// TIA Portal project "conveyer belt system V6.4" (V19)

(* hardware
DEVICE "S71500/ET200MP-Station_1"  S7-1500 station
   slot 0: "Profilschiene_0"  6ES7 590-1***0-0AA0
   slot 1: "PLC_1"  CPU 1511-1 PN  6ES7 511-1AK00-0AB0  V1.8
   slot 2: "AI 8xU/I/RTD/TC ST_1"  AI 8xU/I/RTD/TC ST  6ES7 531-7KF00-0AB0  V2.0
   slot 3: "AI 8xU/I/RTD/TC ST_2"  AI 8xU/I/RTD/TC ST  6ES7 531-7KF00-0AB0  V2.0
   slot 4: "AI 8xU/I/RTD/TC ST_3"  AI 8xU/I/RTD/TC ST  6ES7 531-7KF00-0AB0  V2.0
   slot 5: "AI 8xU/I/RTD/TC ST_4"  AI 8xU/I/RTD/TC ST  6ES7 531-7KF00-0AB0  V2.0
   slot 6: "DI 16x24VDC BA_1"  DI 16x24VDC BA  6ES7 521-1BH10-0AA0  V1.0
DEVICE "HMI_1"  KTP1200 Basic PN
   slot 0: "HMI_1"  KTP1200 Basic PN  6AV2 123-2MB03-0AX0  17.0.0.0
   slot 1: "HMI_RT_2"  KTP1200 Basic PN  6AV2 123-2MB03-0AX0  17.0.0.0
   slot 5: "HMI_1.IE_CP_1"  PROFINET Interface  17.0.0.0
      slot 1: "PROFINET Interface_1"  PROFINET Interface
         slot 1: "Port_1"  Port
*)

// ===== PLC "PLC_1"  CPU 1511-1 PN =====

VAR_GLOBAL   // PLC tag table "Standard-Variablentabelle"
   "Tag_1" AT %I1000.0 : Bool;
   "Tag_2" AT %Q1000.0 : Bool;
   "Tag_3" AT %I1000.1 : Bool;
END_VAR

VAR_GLOBAL   // PLC tag table "control panel"
   "start_button" AT %I0.0 : Bool;
   "reset_button" AT %I0.1 : Bool;
   "stop_button" AT %I0.2 : Bool;
   "emergency_stop" AT %I0.3 : Bool;
   "start_button_light" AT %Q0.0 : Bool;
   "reset_button_light" AT %Q0.1 : Bool;
   "stop_button_light" AT %Q0.2 : Bool;
   "system_start" AT %Q0.3 : Bool;
   "system_fault" AT %Q0.4 : Bool;
   "system_stop" AT %Q0.5 : Bool;
   "sensor_start" AT %I0.7 : Bool;
   "low_power_mode" AT %I0.4 : Bool;
   "sensor_carousel" AT %I1.0 : Bool;
   "carousel_on" AT %I0.5 : Bool;
END_VAR

VAR_GLOBAL   // PLC tag table "conveyor 0"
   "motor+(0)" AT %Q3.7 : Bool;
   "motor-(0)" AT %Q3.6 : Bool;
   "encoder_A(0)" AT %I3.7 : Bool;
   "encoder_B(0)" AT %I3.6 : Bool;
   "sensor(0)" AT %I5.7 : Bool;
END_VAR

VAR_GLOBAL   // PLC tag table "conveyor 1"
   "motor+(1)" AT %Q3.5 : Bool;
   "motor-(1)" AT %Q3.4 : Bool;
   "encoder_A(1)" AT %I3.5 : Bool;
   "encoder_B(1)" AT %I3.4 : Bool;
   "sensor(1)" AT %I5.6 : Bool;
END_VAR

VAR_GLOBAL   // PLC tag table "conveyor 2"
   "motor+(2)" AT %Q3.3 : Bool;
   "motor-(2)" AT %Q3.2 : Bool;
   "encoder_A(2)" AT %I3.3 : Bool;
   "encoder_B(2)" AT %I3.2 : Bool;
   "sensor(2)" AT %I5.5 : Bool;
END_VAR

VAR_GLOBAL   // PLC tag table "conveyor 3"
   "motor+(3)" AT %Q3.1 : Bool;
   "motor-(3)" AT %Q3.0 : Bool;
   "encoder_A(3)" AT %I3.1 : Bool;
   "encoder_B(3)" AT %I3.0 : Bool;
   "sensor(3)" AT %I5.4 : Bool;
END_VAR

VAR_GLOBAL   // PLC tag table "conveyor 4"
   "motor+(4)" AT %Q2.7 : Bool;
   "motor-(4)" AT %Q2.6 : Bool;
   "encoder_A(4)" AT %I2.7 : Bool;
   "encoder_B(4)" AT %I2.6 : Bool;
   "sensor(4)" AT %I5.3 : Bool;
END_VAR

VAR_GLOBAL   // PLC tag table "conveyor 5"
   "motor+(5)" AT %Q2.5 : Bool;
   "motor-(5)" AT %Q2.4 : Bool;
   "encoder_A(5)" AT %I2.5 : Bool;
   "encoder_B(5)" AT %I2.4 : Bool;
   "sensor(5)" AT %I5.2 : Bool;
END_VAR

VAR_GLOBAL   // PLC tag table "conveyor 6"
   "motor+(6)" AT %Q2.3 : Bool;
   "motor-(6)" AT %Q2.2 : Bool;
   "encoder_A(6)" AT %I2.3 : Bool;
   "encoder_B(6)" AT %I2.2 : Bool;
   "sensor(6)" AT %I5.1 : Bool;
END_VAR

DATA_BLOCK "conveyor_0"   // DB1
{ S7_Optimized_Access := 'TRUE' }
VERSION : 0.1
// stored: InstanceOfName conveyor_control
"conveyor_control"
BEGIN
END_DATA_BLOCK

DATA_BLOCK "conveyor_2"   // DB3
{ S7_Optimized_Access := 'TRUE' }
VERSION : 0.1
// stored: InstanceOfName conveyor_control
"conveyor_control"
BEGIN
END_DATA_BLOCK

DATA_BLOCK "conveyor_1"   // DB5
{ S7_Optimized_Access := 'TRUE' }
VERSION : 0.1
// stored: InstanceOfName conveyor_control
"conveyor_control"
BEGIN
END_DATA_BLOCK

DATA_BLOCK "system_control_DB"   // DB6
{ S7_Optimized_Access := 'TRUE' }
VERSION : 0.1
// stored: InstanceOfName system_control
"system_control"
BEGIN
END_DATA_BLOCK

DATA_BLOCK "lamp control_DB"   // DB11
{ S7_Optimized_Access := 'TRUE' }
VERSION : 0.1
// stored: InstanceOfName lamp_control
"lamp_control"
BEGIN
END_DATA_BLOCK

DATA_BLOCK "conveyor_3"   // DB15
{ S7_Optimized_Access := 'TRUE' }
VERSION : 0.1
// stored: InstanceOfName conveyor_control
"conveyor_control"
BEGIN
END_DATA_BLOCK

DATA_BLOCK "conveyor_4"   // DB17
{ S7_Optimized_Access := 'TRUE' }
VERSION : 0.1
// stored: InstanceOfName conveyor_control
"conveyor_control"
BEGIN
END_DATA_BLOCK

DATA_BLOCK "conveyor_5"   // DB19
{ S7_Optimized_Access := 'TRUE' }
VERSION : 0.1
// stored: InstanceOfName conveyor_control
"conveyor_control"
BEGIN
END_DATA_BLOCK

DATA_BLOCK "conveyor_6"   // DB21
{ S7_Optimized_Access := 'TRUE' }
VERSION : 0.1
// stored: InstanceOfName conveyor_control
"conveyor_control"
BEGIN
END_DATA_BLOCK

DATA_BLOCK "standard_parameters"   // DB26
{ S7_Optimized_Access := 'TRUE' }
VERSION : 0.1
   VAR
      "2 meter belt clearance delay" : Time := T#4S;   // need to change to 10s
      "4 meter belt clearance delay" : Time := T#8S;   // need to change to 20s
      "6 meter belt clearance delay" : Time := T#12S;   // need to change to 30s
      "curved belt clearance delay" : Time := T#4S;   // need to change to 10s
   END_VAR
BEGIN
END_DATA_BLOCK

DATA_BLOCK "system_state"   // DB27
{ S7_Optimized_Access := 'TRUE' }
VERSION : 0.1
   VAR
      start_0 : Bool;
      start_1 : Bool;
      all_conveyors_running : Bool;
      some_conveyors_running : Bool;
      "system_start/stop_memory" : Bool;
      fault_flag : Bool;
      low_power_mode : Bool;
      safety_delay : Time;
   END_VAR
BEGIN
END_DATA_BLOCK

FUNCTION_BLOCK "conveyor_control"   // FB1, FBD
{ S7_Optimized_Access := 'TRUE' }
VERSION : 0.1
   VAR_INPUT
      enable_cascade_control : Bool;
      enable_sensor_control : Bool;
      enable_on_delay : Bool;
      enable_off_delay : Bool;
      encoder_A : Bool;
      encoder_B : Bool;
      fault_feedback_in : Bool;
      fault_reset : Bool;
      preceeding_sensor : Bool;
      off_delay : Time;
      on_delay : Time := T#1S;
   END_VAR
   VAR_OUTPUT
      "motor+" : Bool;
      "motor-" : Bool;
      motor_fault : Bool;
      motor_condition : Int;
      fault_feedback_out : Bool;
      remaining_delay : Time;
      running_feedback : Bool;
   END_VAR
   VAR_IN_OUT
      system_fault_flag : Bool;
   END_VAR
   VAR
      encoder_buffer : TOF_TIME;
      encoder_A_edge : R_TRIG;
      encoder_B_edge : R_TRIG;
      fault_buffer : TON_TIME;
      sensor_control_Instance : "sensor_control";
   END_VAR
   VAR RETAIN
      off_delay_instance : TOF_TIME;
      on_delay_instance : TON_TIME;
   END_VAR
BEGIN

REGION Network 1: sensor control
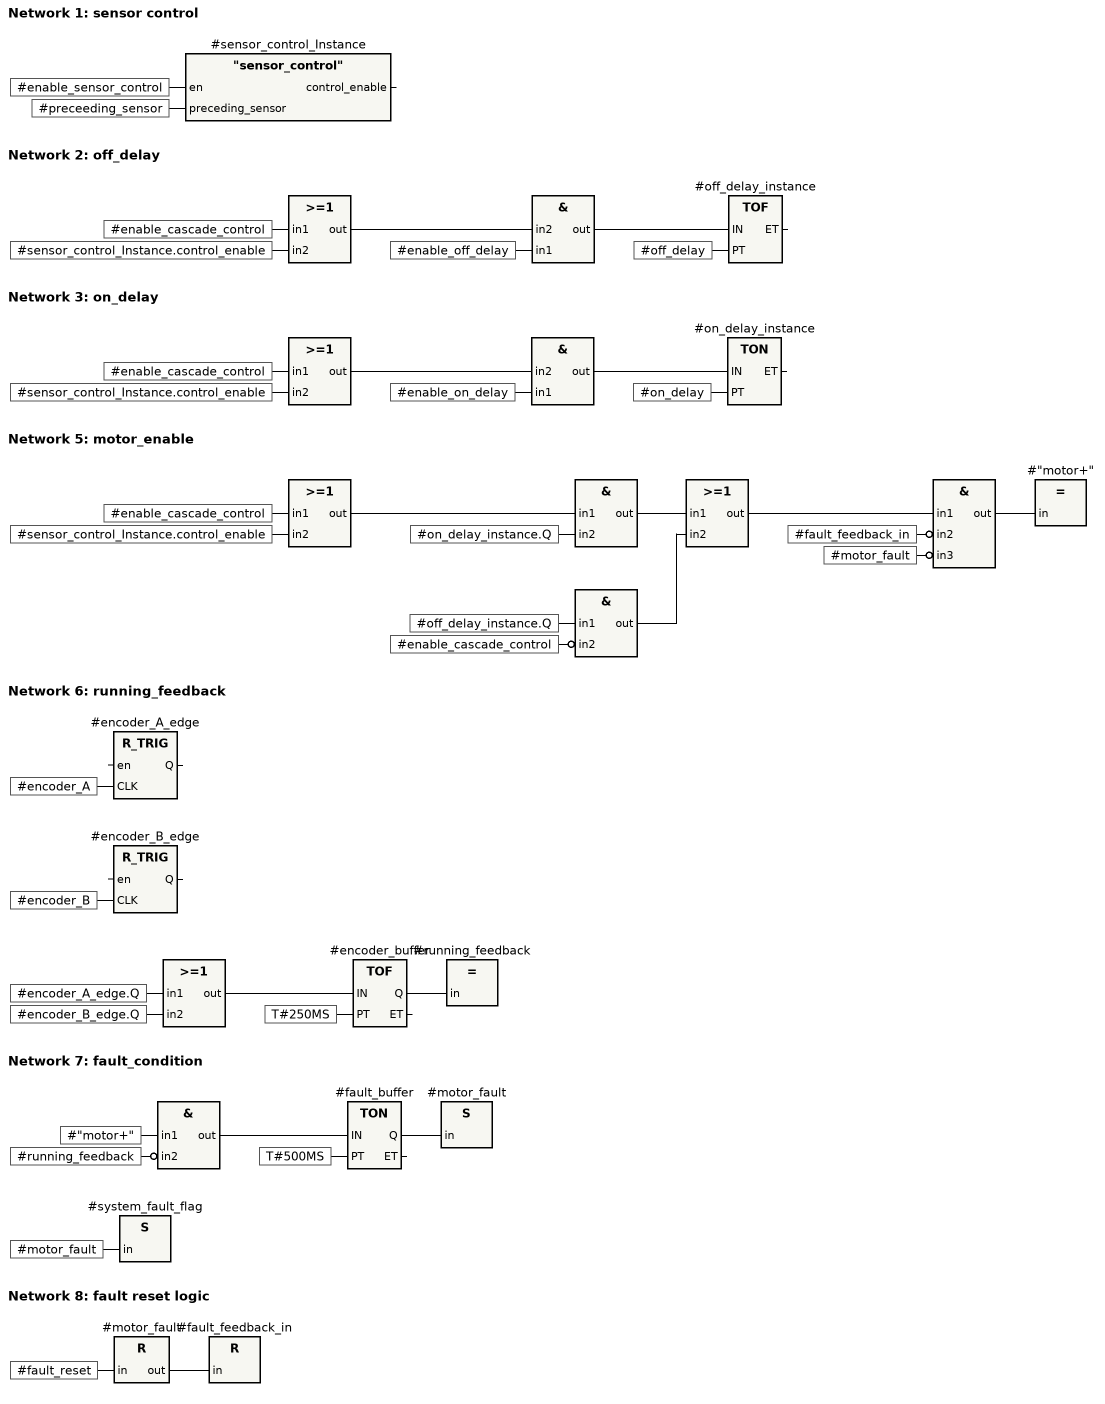
   IF #enable_sensor_control THEN
       #sensor_control_Instance(preceding_sensor := #preceeding_sensor);   // "sensor_control"
   END_IF;
END_REGION

REGION Network 2: off_delay
   #off_delay_instance(IN := (#enable_cascade_control OR #sensor_control_Instance.control_enable) AND #enable_off_delay,   // TOF
                       PT := #off_delay);
END_REGION

REGION Network 3: on_delay
   #on_delay_instance(IN := (#enable_cascade_control OR #sensor_control_Instance.control_enable) AND #enable_on_delay,   // TON
                      PT := #on_delay);
END_REGION

REGION Network 4 (SCL): remaining delay
   IF #enable_off_delay THEN
       #remaining_delay := #off_delay_instance.PT - #off_delay_instance.ET;
   ELSIF #enable_on_delay THEN
       #remaining_delay := #on_delay_instance.PT - #on_delay_instance.ET;
   END_IF;
END_REGION

REGION Network 5: motor_enable
   #"motor+" := (((#enable_cascade_control OR #sensor_control_Instance.control_enable) AND #on_delay_instance.Q) OR (#off_delay_instance.Q AND NOT #enable_cascade_control)) AND NOT #fault_feedback_in AND NOT #motor_fault;
END_REGION

REGION Network 6: running_feedback
   #encoder_A_edge(CLK := #encoder_A);   // R_TRIG
   #encoder_B_edge(CLK := #encoder_B);   // R_TRIG
   #encoder_buffer(IN := #encoder_A_edge.Q OR #encoder_B_edge.Q, PT := T#250MS);   // TOF
   #running_feedback := #encoder_buffer.Q;
END_REGION

REGION Network 7: fault_condition
   #fault_buffer(IN := #"motor+" AND NOT #running_feedback, PT := T#500MS);   // TON
   IF #fault_buffer.Q THEN #motor_fault := TRUE; END_IF;
   IF #motor_fault THEN #system_fault_flag := TRUE; END_IF;
END_REGION

REGION Network 8: fault reset logic
   IF #fault_reset THEN
       #motor_fault := FALSE;
       #fault_feedback_in := FALSE;
   END_IF;
END_REGION

REGION Network 9: fault_feedback_loop
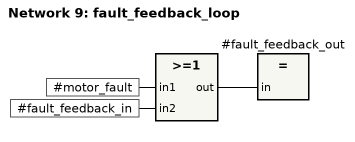
   #fault_feedback_out := #motor_fault OR #fault_feedback_in;
END_REGION

REGION Network 10 (SCL): motor_condition_report
   IF #"motor_fault" THEN
       #"motor_condition" := -1; (*motor fault*)
   ELSIF #"running_feedback" THEN
       #"motor_condition" := 1; (*motor running*)
   ELSIF "system_state".low_power_mode AND NOT #"fault_feedback_in" THEN
       #"motor_condition" := 2; (*low power mode*)
   ELSE
       #"motor_condition" := 0; (*motor stopped*)
   END_IF;
END_REGION
END_FUNCTION_BLOCK

FUNCTION_BLOCK "sensor_control"   // FB2, FBD
{ S7_Optimized_Access := 'TRUE' }
VERSION : 0.1
   VAR_INPUT
      preceding_sensor : Bool;
   END_VAR
   VAR_OUTPUT
      control_enable : Bool;
   END_VAR
   VAR
      sensor_mem_reset_buffer : TOF_TIME;
   END_VAR
   VAR RETAIN
      sensor_memory : Bool;
   END_VAR
BEGIN

REGION Network 1
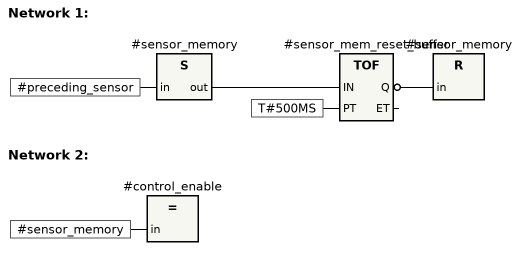
   IF #preceding_sensor THEN #sensor_memory := TRUE; END_IF;
   #sensor_mem_reset_buffer(IN := #preceding_sensor, PT := T#500MS);   // TOF
   IF NOT #sensor_mem_reset_buffer.Q THEN #sensor_memory := FALSE; END_IF;
END_REGION

REGION Network 2
   #control_enable := #sensor_memory;
END_REGION
END_FUNCTION_BLOCK

FUNCTION_BLOCK "lamp_control"   // FB3, FBD
{ S7_Optimized_Access := 'TRUE' }
VERSION : 0.1
   VAR_INPUT
      "start/stop_memory" : Bool;
      all_conveyors_running : Bool;
      conveyors_running : Bool;
      low_power_mode : Bool;
      fault_flag : Bool;
   END_VAR
   VAR_OUTPUT
      start : Bool;
      fault : Bool;
      stop : Bool;
      state : Byte;
   END_VAR
   VAR
      start_pulse : "pulse";
      stop_pulse : "pulse";
      fault_pulse : "pulse";
   END_VAR
BEGIN

REGION Network 1 (SCL): feature debug
   #state := SHL(IN := BOOL_TO_BYTE(#"start/stop_memory"), N := 4) OR
   SHL(IN := BOOL_TO_BYTE(#all_conveyors_running), N := 3) OR
   SHL(IN := BOOL_TO_BYTE(#conveyors_running), N := 2) OR
   SHL(IN := BOOL_TO_BYTE(#low_power_mode), N := 1) OR
   SHL(IN := BOOL_TO_BYTE(#fault_flag), N := 0);
END_REGION

REGION Network 2: start logic
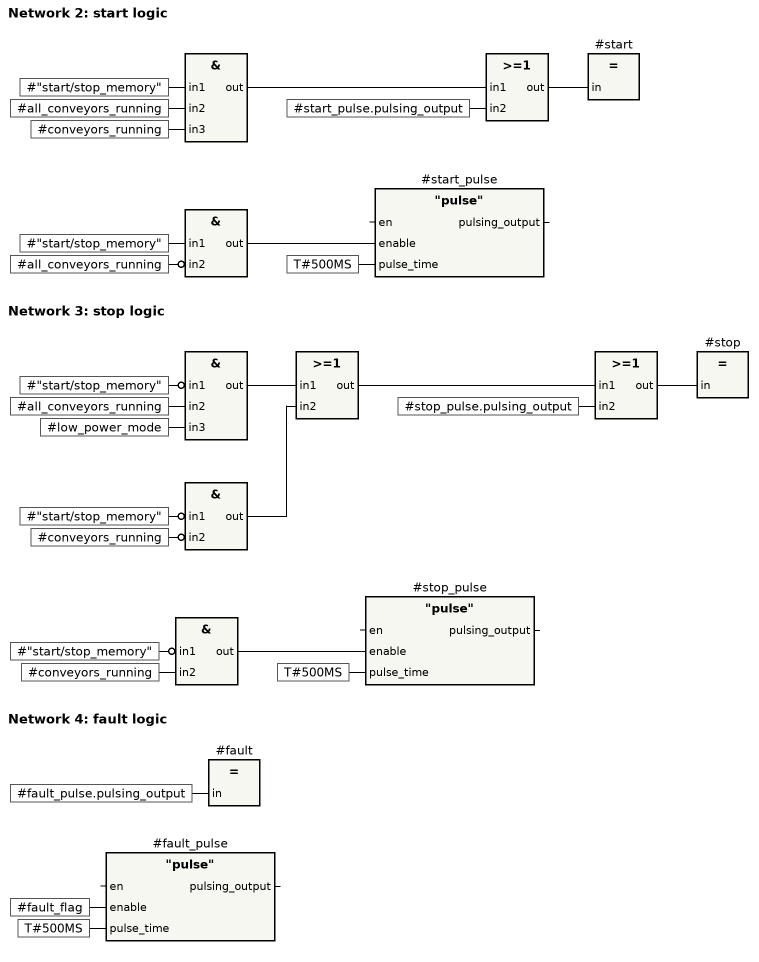
   #start := (#"start/stop_memory" AND #all_conveyors_running AND #conveyors_running) OR #start_pulse.pulsing_output;
   #start_pulse(enable := #"start/stop_memory" AND NOT #all_conveyors_running, pulse_time := T#500MS);   // "pulse"
END_REGION

REGION Network 3: stop logic
   #stop := (NOT #"start/stop_memory" AND #all_conveyors_running AND #low_power_mode) OR (NOT #"start/stop_memory" AND NOT #conveyors_running) OR #stop_pulse.pulsing_output;
   #stop_pulse(enable := NOT #"start/stop_memory" AND #conveyors_running, pulse_time := T#500MS);   // "pulse"
END_REGION

REGION Network 4: fault logic
   #fault := #fault_pulse.pulsing_output;
   #fault_pulse(enable := #fault_flag, pulse_time := T#500MS);   // "pulse"
END_REGION
END_FUNCTION_BLOCK

FUNCTION_BLOCK "pulse"   // FB4, FBD
{ S7_Optimized_Access := 'TRUE' }
VERSION : 0.1
   VAR_INPUT
      enable : Bool;
      pulse_time : Time;
   END_VAR
   VAR_OUTPUT
      pulsing_output : Bool;
   END_VAR
   VAR
      time_delay_bit : Bool;
      IEC_Timer_0_Instance : TON_TIME;
      IEC_Timer_0_Instance_1 : TON_TIME;
   END_VAR
BEGIN

REGION Network 1
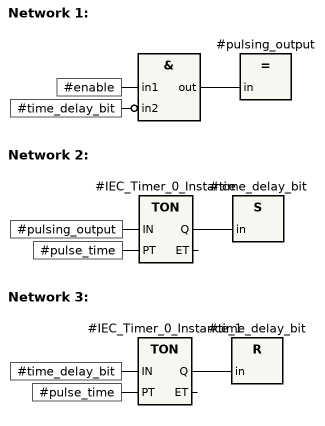
   #pulsing_output := #enable AND NOT #time_delay_bit;
END_REGION

REGION Network 2
   #IEC_Timer_0_Instance(IN := #pulsing_output, PT := #pulse_time);   // TON
   IF #IEC_Timer_0_Instance.Q THEN #time_delay_bit := TRUE; END_IF;
END_REGION

REGION Network 3
   #IEC_Timer_0_Instance_1(IN := #time_delay_bit, PT := #pulse_time);   // TON
   IF #IEC_Timer_0_Instance_1.Q THEN #time_delay_bit := FALSE; END_IF;
END_REGION
END_FUNCTION_BLOCK

FUNCTION_BLOCK "system_control"   // FB5, FBD
{ S7_Optimized_Access := 'TRUE' }
VERSION : 0.1
   VAR_INPUT
      start_button : Bool;
      reset_button : Bool;
      stop_button : Bool;
   END_VAR
   VAR_IN_OUT
      system_fault_flag : Bool;
      "system_start/stop_memory" : Bool;
      system_all_conv_running : Bool;
      system_some_conv_running : Bool;
      system_LP_mode : Bool;
      safety_delay : Time;
   END_VAR
   VAR
      reset_off_delay : TOF_TIME;
      reset_on_delay : TON_TIME;
      start_0 : Bool;
      start_1 : Bool;
      system_start_on_delay : TON_TIME;
      low_power_enable_delay : TON_TIME;
      reset_pulse_1 : TP_TIME;
      reset_pulse_fault : TP_TIME;
      reset_pulse_startstop : TP_TIME;
   END_VAR
   VAR_TEMP   // added for the SCL form of the ladder/FBD networks
      _w1 : Bool;
   END_VAR
BEGIN

REGION Network 1: system state fault reset logic
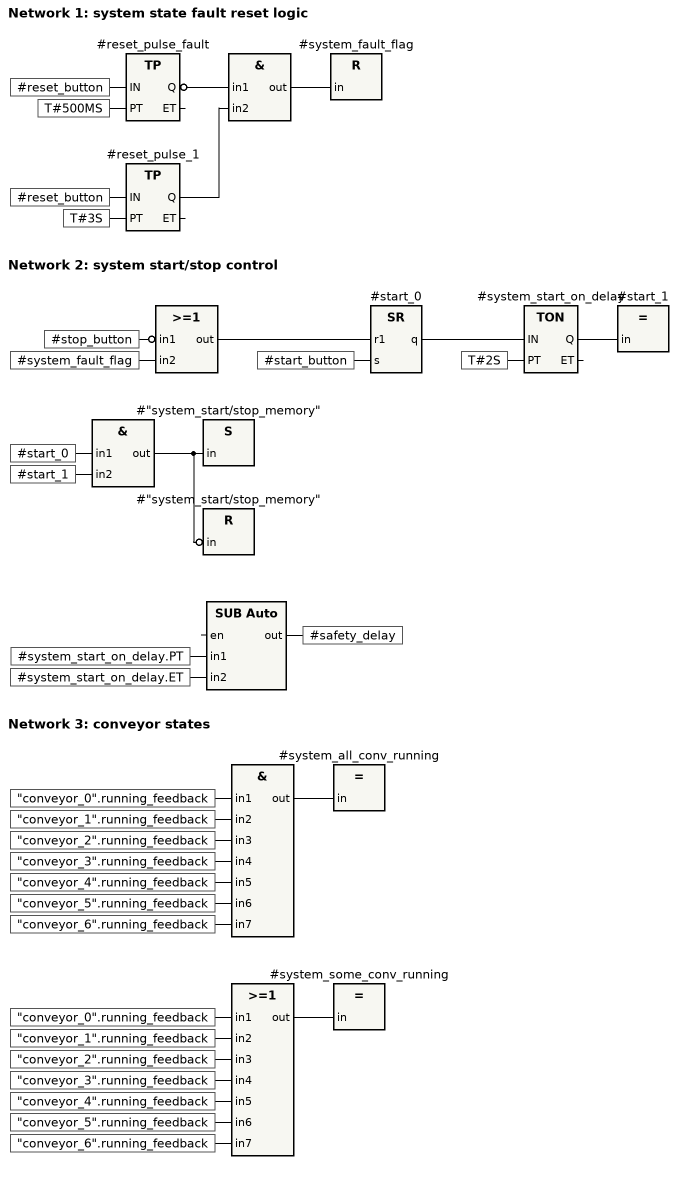
   #reset_pulse_fault(IN := #reset_button, PT := T#500MS);   // TP
   #reset_pulse_1(IN := #reset_button, PT := T#3S);   // TP
   IF NOT #reset_pulse_fault.Q AND #reset_pulse_1.Q THEN #system_fault_flag := FALSE; END_IF;
END_REGION

REGION Network 2: system start/stop control
   IF #start_button THEN
       #start_0 := TRUE;   // SR flip-flop
   END_IF;
   IF NOT #stop_button OR #system_fault_flag THEN #start_0 := FALSE; END_IF;
   #system_start_on_delay(IN := #start_0, PT := T#2S);   // TON
   #start_1 := #system_start_on_delay.Q;
   #_w1 := #start_0 AND #start_1;
   IF #_w1 THEN #"system_start/stop_memory" := TRUE; END_IF;
   IF NOT #_w1 THEN #"system_start/stop_memory" := FALSE; END_IF;
   #safety_delay := #system_start_on_delay.PT - #system_start_on_delay.ET;
END_REGION

REGION Network 3: conveyor states
   #system_all_conv_running := "conveyor_0".running_feedback AND "conveyor_1".running_feedback AND "conveyor_2".running_feedback AND "conveyor_3".running_feedback AND "conveyor_4".running_feedback AND "conveyor_5".running_feedback AND "conveyor_6".running_feedback;
   #system_some_conv_running := "conveyor_0".running_feedback OR "conveyor_1".running_feedback OR "conveyor_2".running_feedback OR "conveyor_3".running_feedback OR "conveyor_4".running_feedback OR "conveyor_5".running_feedback OR "conveyor_6".running_feedback;
END_REGION

REGION Network 4: low power logic
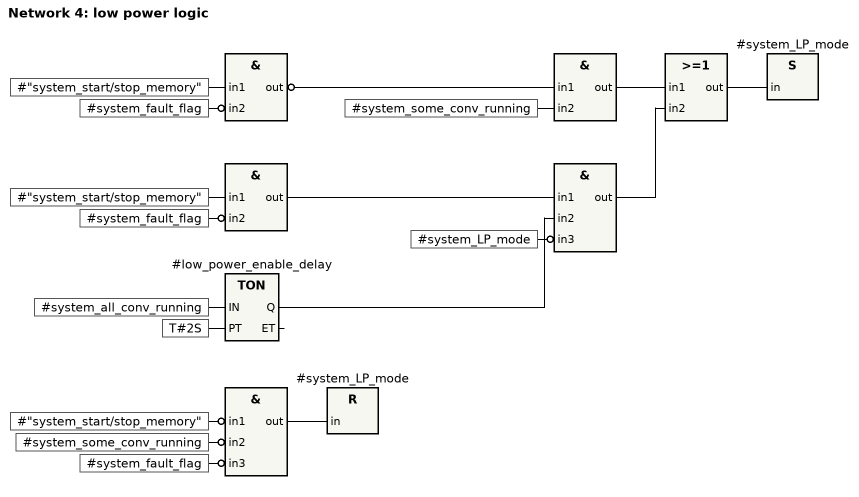
   #low_power_enable_delay(IN := #system_all_conv_running, PT := T#2S);   // TON
   IF (NOT (#"system_start/stop_memory" AND NOT #system_fault_flag) AND #system_some_conv_running) OR (#"system_start/stop_memory" AND NOT #system_fault_flag AND #low_power_enable_delay.Q AND NOT #system_LP_mode) THEN
       #system_LP_mode := TRUE;
   END_IF;
   IF NOT #"system_start/stop_memory" AND NOT #system_some_conv_running AND NOT #system_fault_flag THEN
       #system_LP_mode := FALSE;
   END_IF;
END_REGION
END_FUNCTION_BLOCK

FUNCTION "main_loop" : Void   // FC1, FBD
{ S7_Optimized_Access := 'TRUE' }
VERSION : 0.1
BEGIN

REGION Network 1
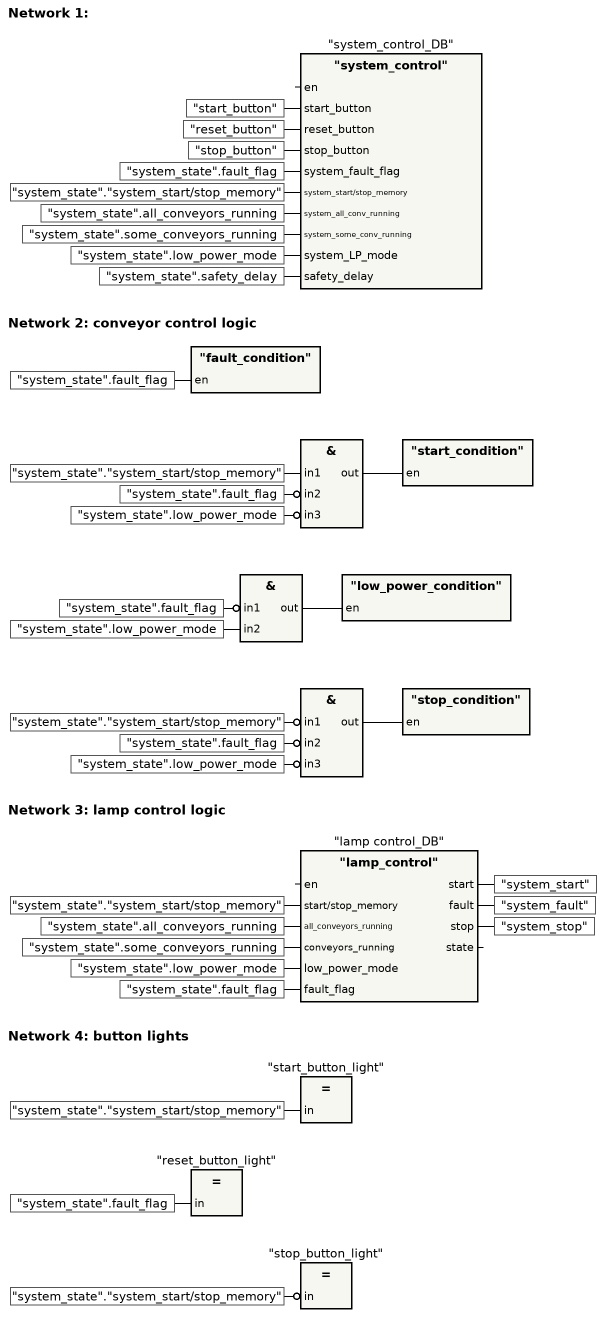
   "system_control_DB"(start_button := "start_button",   // "system_control"
                       reset_button := "reset_button",
                       stop_button := "stop_button",
                       system_fault_flag := "system_state".fault_flag,
                       "system_start/stop_memory" := "system_state"."system_start/stop_memory",
                       system_all_conv_running := "system_state".all_conveyors_running,
                       system_some_conv_running := "system_state".some_conveyors_running,
                       system_LP_mode := "system_state".low_power_mode,
                       safety_delay := "system_state".safety_delay);
END_REGION

REGION Network 2: conveyor control logic
   IF "system_state".fault_flag THEN "fault_condition"(); END_IF;
   IF "system_state"."system_start/stop_memory" AND NOT "system_state".fault_flag AND NOT "system_state".low_power_mode THEN
       "start_condition"();
   END_IF;
   IF NOT "system_state".fault_flag AND "system_state".low_power_mode THEN "low_power_condition"(); END_IF;
   IF NOT "system_state"."system_start/stop_memory" AND NOT "system_state".fault_flag AND NOT "system_state".low_power_mode THEN
       "stop_condition"();
   END_IF;
END_REGION

REGION Network 3: lamp control logic
   "lamp control_DB"("start/stop_memory" := "system_state"."system_start/stop_memory",   // "lamp_control"
                     all_conveyors_running := "system_state".all_conveyors_running,
                     conveyors_running := "system_state".some_conveyors_running,
                     low_power_mode := "system_state".low_power_mode,
                     fault_flag := "system_state".fault_flag,
                     start => "system_start",
                     fault => "system_fault",
                     stop => "system_stop");
END_REGION

REGION Network 4: button lights
   "start_button_light" := "system_state"."system_start/stop_memory";
   "reset_button_light" := "system_state".fault_flag;
   "stop_button_light" := NOT "system_state"."system_start/stop_memory";
END_REGION
END_FUNCTION

FUNCTION "start_condition" : Void   // FC2, FBD
{ S7_Optimized_Access := 'TRUE' }
VERSION : 0.1
BEGIN

REGION Network 1
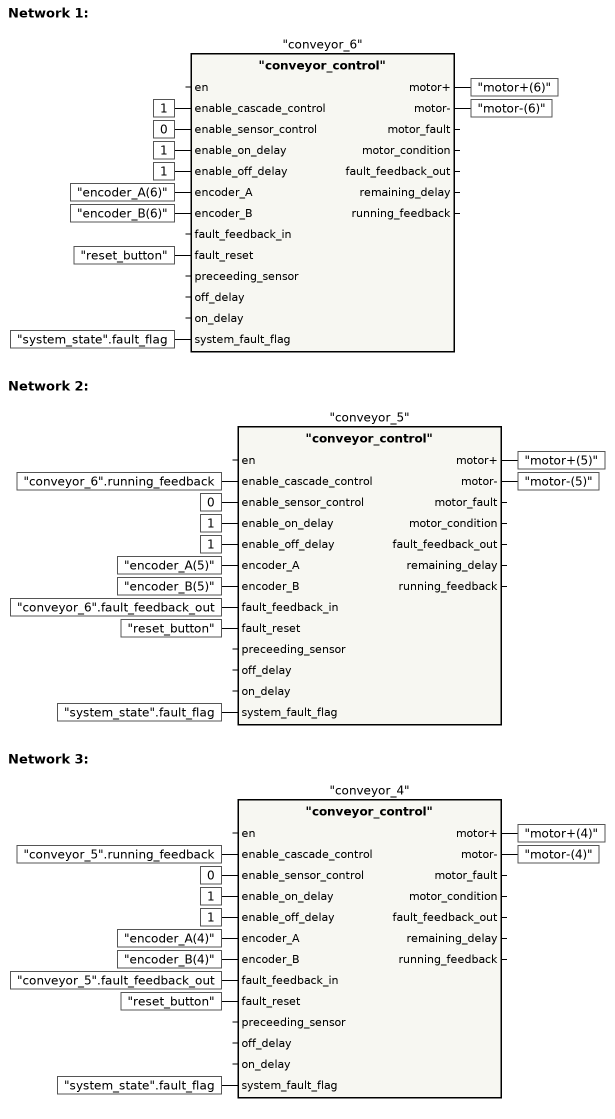
   "conveyor_6"(enable_cascade_control := 1,   // "conveyor_control"
                enable_sensor_control := 0,
                enable_on_delay := 1,
                enable_off_delay := 1,
                encoder_A := "encoder_A(6)",
                encoder_B := "encoder_B(6)",
                fault_reset := "reset_button",
                system_fault_flag := "system_state".fault_flag,
                "motor+" => "motor+(6)",
                "motor-" => "motor-(6)");
END_REGION

REGION Network 2
   "conveyor_5"(enable_cascade_control := "conveyor_6".running_feedback,   // "conveyor_control"
                enable_sensor_control := 0,
                enable_on_delay := 1,
                enable_off_delay := 1,
                encoder_A := "encoder_A(5)",
                encoder_B := "encoder_B(5)",
                fault_feedback_in := "conveyor_6".fault_feedback_out,
                fault_reset := "reset_button",
                system_fault_flag := "system_state".fault_flag,
                "motor+" => "motor+(5)",
                "motor-" => "motor-(5)");
END_REGION

REGION Network 3
   "conveyor_4"(enable_cascade_control := "conveyor_5".running_feedback,   // "conveyor_control"
                enable_sensor_control := 0,
                enable_on_delay := 1,
                enable_off_delay := 1,
                encoder_A := "encoder_A(4)",
                encoder_B := "encoder_B(4)",
                fault_feedback_in := "conveyor_5".fault_feedback_out,
                fault_reset := "reset_button",
                system_fault_flag := "system_state".fault_flag,
                "motor+" => "motor+(4)",
                "motor-" => "motor-(4)");
END_REGION

REGION Network 4
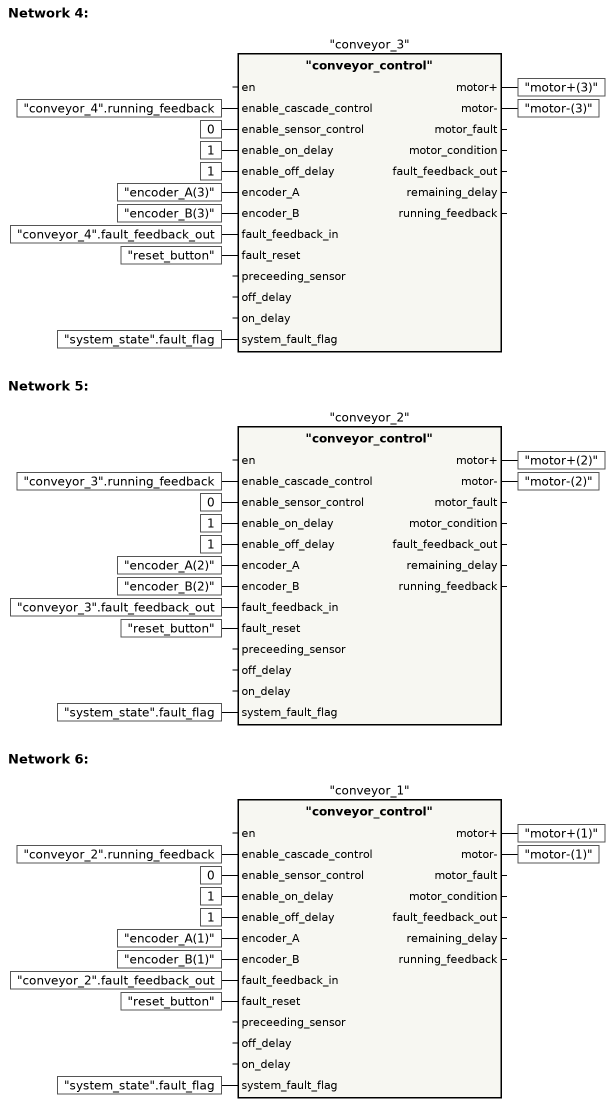
   "conveyor_3"(enable_cascade_control := "conveyor_4".running_feedback,   // "conveyor_control"
                enable_sensor_control := 0,
                enable_on_delay := 1,
                enable_off_delay := 1,
                encoder_A := "encoder_A(3)",
                encoder_B := "encoder_B(3)",
                fault_feedback_in := "conveyor_4".fault_feedback_out,
                fault_reset := "reset_button",
                system_fault_flag := "system_state".fault_flag,
                "motor+" => "motor+(3)",
                "motor-" => "motor-(3)");
END_REGION

REGION Network 5
   "conveyor_2"(enable_cascade_control := "conveyor_3".running_feedback,   // "conveyor_control"
                enable_sensor_control := 0,
                enable_on_delay := 1,
                enable_off_delay := 1,
                encoder_A := "encoder_A(2)",
                encoder_B := "encoder_B(2)",
                fault_feedback_in := "conveyor_3".fault_feedback_out,
                fault_reset := "reset_button",
                system_fault_flag := "system_state".fault_flag,
                "motor+" => "motor+(2)",
                "motor-" => "motor-(2)");
END_REGION

REGION Network 6
   "conveyor_1"(enable_cascade_control := "conveyor_2".running_feedback,   // "conveyor_control"
                enable_sensor_control := 0,
                enable_on_delay := 1,
                enable_off_delay := 1,
                encoder_A := "encoder_A(1)",
                encoder_B := "encoder_B(1)",
                fault_feedback_in := "conveyor_2".fault_feedback_out,
                fault_reset := "reset_button",
                system_fault_flag := "system_state".fault_flag,
                "motor+" => "motor+(1)",
                "motor-" => "motor-(1)");
END_REGION

REGION Network 7
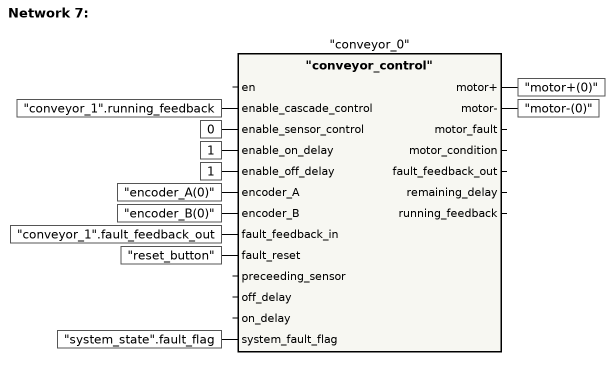
   "conveyor_0"(enable_cascade_control := "conveyor_1".running_feedback,   // "conveyor_control"
                enable_sensor_control := 0,
                enable_on_delay := 1,
                enable_off_delay := 1,
                encoder_A := "encoder_A(0)",
                encoder_B := "encoder_B(0)",
                fault_feedback_in := "conveyor_1".fault_feedback_out,
                fault_reset := "reset_button",
                system_fault_flag := "system_state".fault_flag,
                "motor+" => "motor+(0)",
                "motor-" => "motor-(0)");
END_REGION
END_FUNCTION

FUNCTION "stop_condition" : Void   // FC3, FBD
{ S7_Optimized_Access := 'TRUE' }
VERSION : 0.1
BEGIN

REGION Network 1
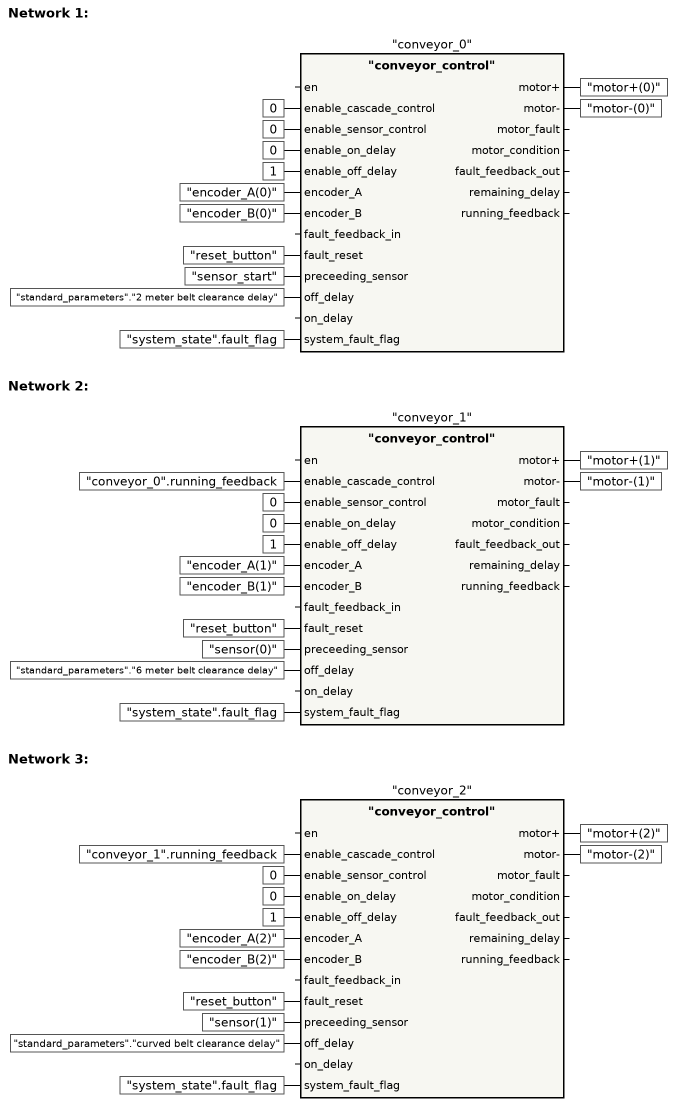
   "conveyor_0"(enable_cascade_control := 0,   // "conveyor_control"
                enable_sensor_control := 0,
                enable_on_delay := 0,
                enable_off_delay := 1,
                encoder_A := "encoder_A(0)",
                encoder_B := "encoder_B(0)",
                fault_reset := "reset_button",
                preceeding_sensor := "sensor_start",
                off_delay := "standard_parameters"."2 meter belt clearance delay",
                system_fault_flag := "system_state".fault_flag,
                "motor+" => "motor+(0)",
                "motor-" => "motor-(0)");
END_REGION

REGION Network 2
   "conveyor_1"(enable_cascade_control := "conveyor_0".running_feedback,   // "conveyor_control"
                enable_sensor_control := 0,
                enable_on_delay := 0,
                enable_off_delay := 1,
                encoder_A := "encoder_A(1)",
                encoder_B := "encoder_B(1)",
                fault_reset := "reset_button",
                preceeding_sensor := "sensor(0)",
                off_delay := "standard_parameters"."6 meter belt clearance delay",
                system_fault_flag := "system_state".fault_flag,
                "motor+" => "motor+(1)",
                "motor-" => "motor-(1)");
END_REGION

REGION Network 3
   "conveyor_2"(enable_cascade_control := "conveyor_1".running_feedback,   // "conveyor_control"
                enable_sensor_control := 0,
                enable_on_delay := 0,
                enable_off_delay := 1,
                encoder_A := "encoder_A(2)",
                encoder_B := "encoder_B(2)",
                fault_reset := "reset_button",
                preceeding_sensor := "sensor(1)",
                off_delay := "standard_parameters"."curved belt clearance delay",
                system_fault_flag := "system_state".fault_flag,
                "motor+" => "motor+(2)",
                "motor-" => "motor-(2)");
END_REGION

REGION Network 4
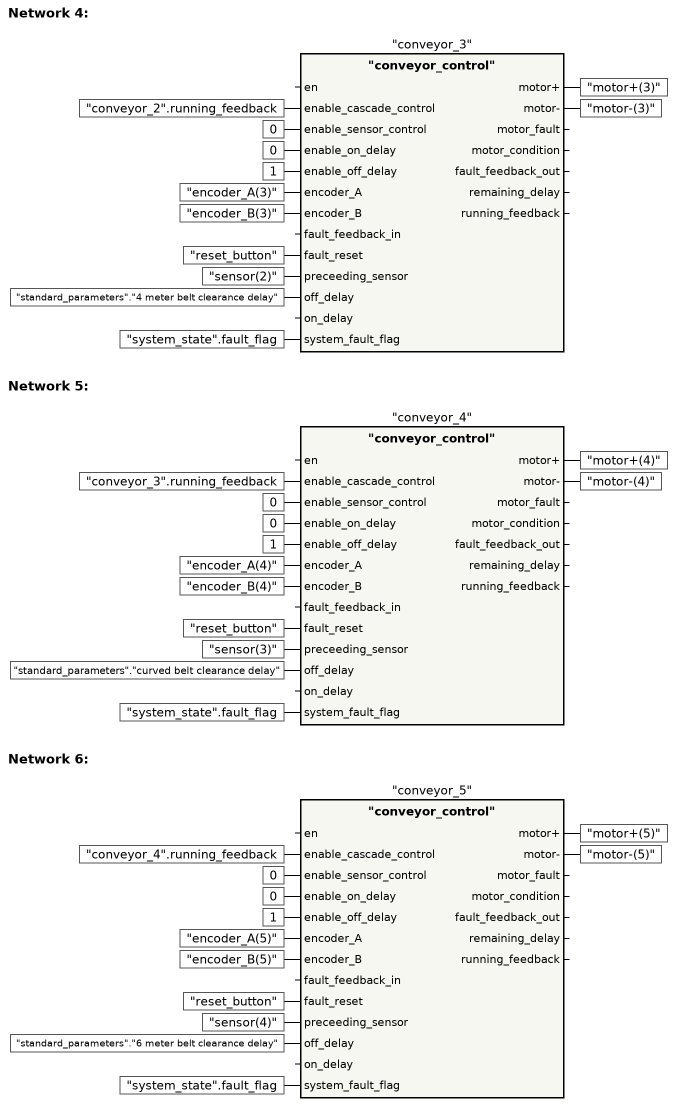
   "conveyor_3"(enable_cascade_control := "conveyor_2".running_feedback,   // "conveyor_control"
                enable_sensor_control := 0,
                enable_on_delay := 0,
                enable_off_delay := 1,
                encoder_A := "encoder_A(3)",
                encoder_B := "encoder_B(3)",
                fault_reset := "reset_button",
                preceeding_sensor := "sensor(2)",
                off_delay := "standard_parameters"."4 meter belt clearance delay",
                system_fault_flag := "system_state".fault_flag,
                "motor+" => "motor+(3)",
                "motor-" => "motor-(3)");
END_REGION

REGION Network 5
   "conveyor_4"(enable_cascade_control := "conveyor_3".running_feedback,   // "conveyor_control"
                enable_sensor_control := 0,
                enable_on_delay := 0,
                enable_off_delay := 1,
                encoder_A := "encoder_A(4)",
                encoder_B := "encoder_B(4)",
                fault_reset := "reset_button",
                preceeding_sensor := "sensor(3)",
                off_delay := "standard_parameters"."curved belt clearance delay",
                system_fault_flag := "system_state".fault_flag,
                "motor+" => "motor+(4)",
                "motor-" => "motor-(4)");
END_REGION

REGION Network 6
   "conveyor_5"(enable_cascade_control := "conveyor_4".running_feedback,   // "conveyor_control"
                enable_sensor_control := 0,
                enable_on_delay := 0,
                enable_off_delay := 1,
                encoder_A := "encoder_A(5)",
                encoder_B := "encoder_B(5)",
                fault_reset := "reset_button",
                preceeding_sensor := "sensor(4)",
                off_delay := "standard_parameters"."6 meter belt clearance delay",
                system_fault_flag := "system_state".fault_flag,
                "motor+" => "motor+(5)",
                "motor-" => "motor-(5)");
END_REGION

REGION Network 7
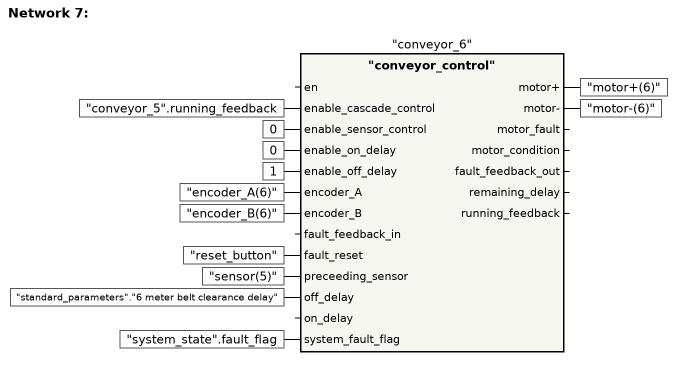
   "conveyor_6"(enable_cascade_control := "conveyor_5".running_feedback,   // "conveyor_control"
                enable_sensor_control := 0,
                enable_on_delay := 0,
                enable_off_delay := 1,
                encoder_A := "encoder_A(6)",
                encoder_B := "encoder_B(6)",
                fault_reset := "reset_button",
                preceeding_sensor := "sensor(5)",
                off_delay := "standard_parameters"."6 meter belt clearance delay",
                system_fault_flag := "system_state".fault_flag,
                "motor+" => "motor+(6)",
                "motor-" => "motor-(6)");
END_REGION
END_FUNCTION

FUNCTION "low_power_condition" : Void   // FC4, FBD
{ S7_Optimized_Access := 'TRUE' }
VERSION : 0.1
BEGIN

REGION Network 1
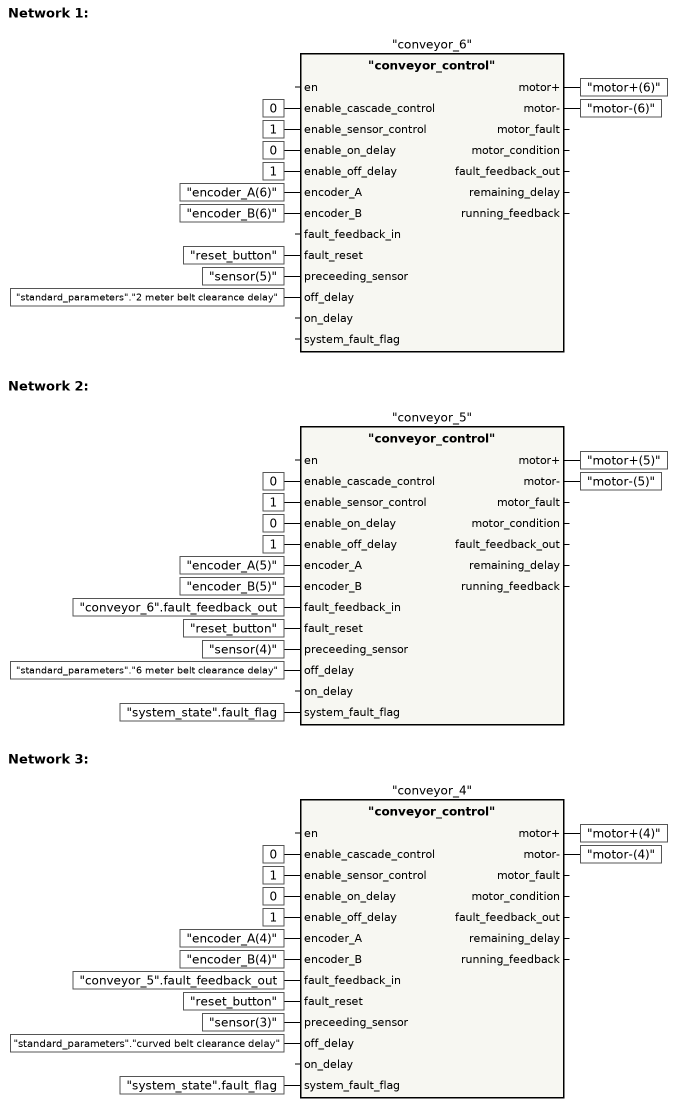
   "conveyor_6"(enable_cascade_control := 0,   // "conveyor_control"
                enable_sensor_control := 1,
                enable_on_delay := 0,
                enable_off_delay := 1,
                encoder_A := "encoder_A(6)",
                encoder_B := "encoder_B(6)",
                fault_reset := "reset_button",
                preceeding_sensor := "sensor(5)",
                off_delay := "standard_parameters"."2 meter belt clearance delay",
                "motor+" => "motor+(6)",
                "motor-" => "motor-(6)");
END_REGION

REGION Network 2
   "conveyor_5"(enable_cascade_control := 0,   // "conveyor_control"
                enable_sensor_control := 1,
                enable_on_delay := 0,
                enable_off_delay := 1,
                encoder_A := "encoder_A(5)",
                encoder_B := "encoder_B(5)",
                fault_feedback_in := "conveyor_6".fault_feedback_out,
                fault_reset := "reset_button",
                preceeding_sensor := "sensor(4)",
                off_delay := "standard_parameters"."6 meter belt clearance delay",
                system_fault_flag := "system_state".fault_flag,
                "motor+" => "motor+(5)",
                "motor-" => "motor-(5)");
END_REGION

REGION Network 3
   "conveyor_4"(enable_cascade_control := 0,   // "conveyor_control"
                enable_sensor_control := 1,
                enable_on_delay := 0,
                enable_off_delay := 1,
                encoder_A := "encoder_A(4)",
                encoder_B := "encoder_B(4)",
                fault_feedback_in := "conveyor_5".fault_feedback_out,
                fault_reset := "reset_button",
                preceeding_sensor := "sensor(3)",
                off_delay := "standard_parameters"."curved belt clearance delay",
                system_fault_flag := "system_state".fault_flag,
                "motor+" => "motor+(4)",
                "motor-" => "motor-(4)");
END_REGION

REGION Network 4
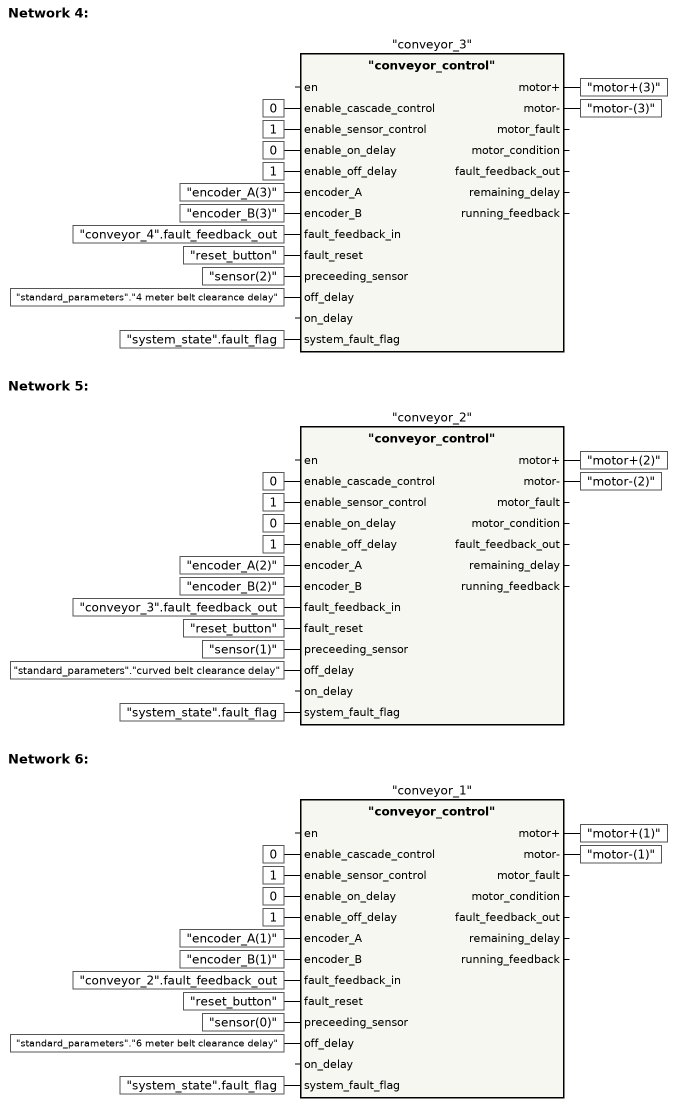
   "conveyor_3"(enable_cascade_control := 0,   // "conveyor_control"
                enable_sensor_control := 1,
                enable_on_delay := 0,
                enable_off_delay := 1,
                encoder_A := "encoder_A(3)",
                encoder_B := "encoder_B(3)",
                fault_feedback_in := "conveyor_4".fault_feedback_out,
                fault_reset := "reset_button",
                preceeding_sensor := "sensor(2)",
                off_delay := "standard_parameters"."4 meter belt clearance delay",
                system_fault_flag := "system_state".fault_flag,
                "motor+" => "motor+(3)",
                "motor-" => "motor-(3)");
END_REGION

REGION Network 5
   "conveyor_2"(enable_cascade_control := 0,   // "conveyor_control"
                enable_sensor_control := 1,
                enable_on_delay := 0,
                enable_off_delay := 1,
                encoder_A := "encoder_A(2)",
                encoder_B := "encoder_B(2)",
                fault_feedback_in := "conveyor_3".fault_feedback_out,
                fault_reset := "reset_button",
                preceeding_sensor := "sensor(1)",
                off_delay := "standard_parameters"."curved belt clearance delay",
                system_fault_flag := "system_state".fault_flag,
                "motor+" => "motor+(2)",
                "motor-" => "motor-(2)");
END_REGION

REGION Network 6
   "conveyor_1"(enable_cascade_control := 0,   // "conveyor_control"
                enable_sensor_control := 1,
                enable_on_delay := 0,
                enable_off_delay := 1,
                encoder_A := "encoder_A(1)",
                encoder_B := "encoder_B(1)",
                fault_feedback_in := "conveyor_2".fault_feedback_out,
                fault_reset := "reset_button",
                preceeding_sensor := "sensor(0)",
                off_delay := "standard_parameters"."6 meter belt clearance delay",
                system_fault_flag := "system_state".fault_flag,
                "motor+" => "motor+(1)",
                "motor-" => "motor-(1)");
END_REGION

REGION Network 7
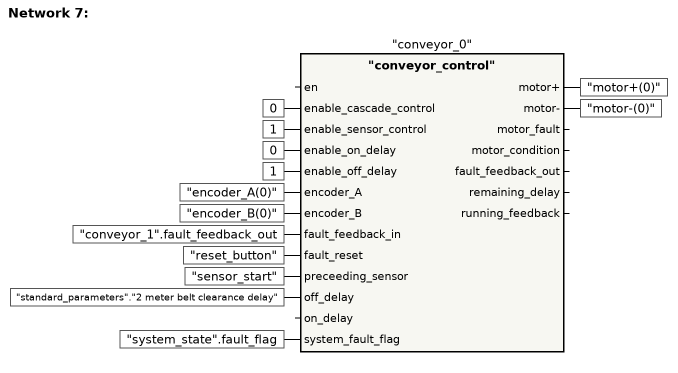
   "conveyor_0"(enable_cascade_control := 0,   // "conveyor_control"
                enable_sensor_control := 1,
                enable_on_delay := 0,
                enable_off_delay := 1,
                encoder_A := "encoder_A(0)",
                encoder_B := "encoder_B(0)",
                fault_feedback_in := "conveyor_1".fault_feedback_out,
                fault_reset := "reset_button",
                preceeding_sensor := "sensor_start",
                off_delay := "standard_parameters"."2 meter belt clearance delay",
                system_fault_flag := "system_state".fault_flag,
                "motor+" => "motor+(0)",
                "motor-" => "motor-(0)");
END_REGION
END_FUNCTION

FUNCTION "fault_condition" : Void   // FC5, FBD
{ S7_Optimized_Access := 'TRUE' }
VERSION : 0.1
BEGIN

REGION Network 1
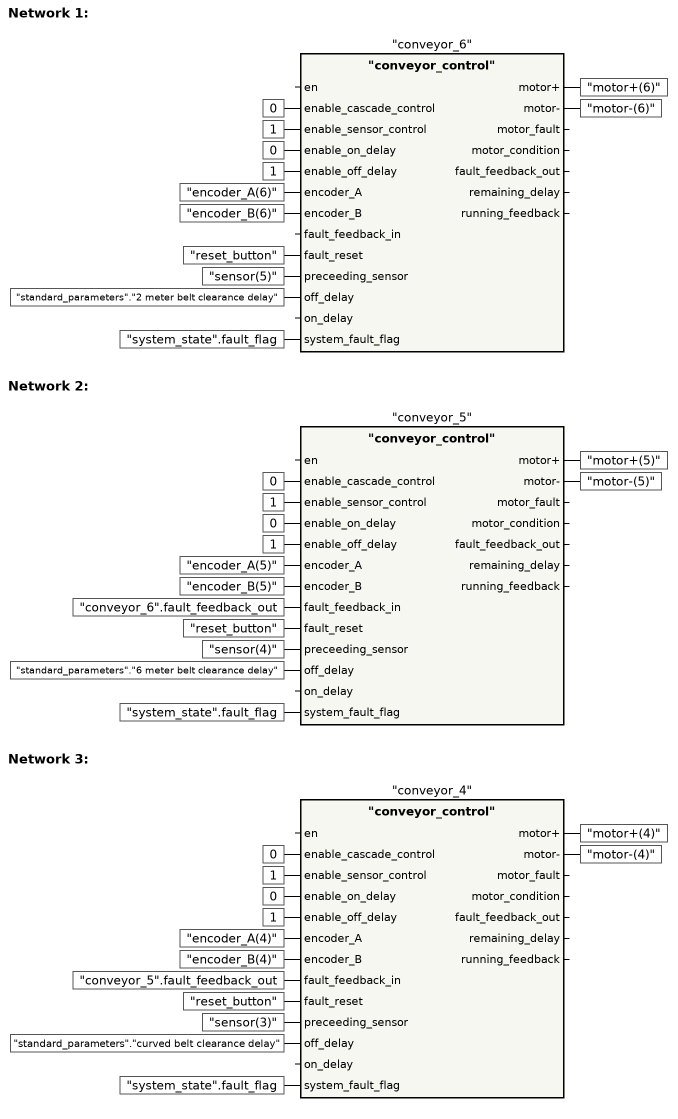
   "conveyor_6"(enable_cascade_control := 0,   // "conveyor_control"
                enable_sensor_control := 1,
                enable_on_delay := 0,
                enable_off_delay := 1,
                encoder_A := "encoder_A(6)",
                encoder_B := "encoder_B(6)",
                fault_reset := "reset_button",
                preceeding_sensor := "sensor(5)",
                off_delay := "standard_parameters"."2 meter belt clearance delay",
                system_fault_flag := "system_state".fault_flag,
                "motor+" => "motor+(6)",
                "motor-" => "motor-(6)");
END_REGION

REGION Network 2
   "conveyor_5"(enable_cascade_control := 0,   // "conveyor_control"
                enable_sensor_control := 1,
                enable_on_delay := 0,
                enable_off_delay := 1,
                encoder_A := "encoder_A(5)",
                encoder_B := "encoder_B(5)",
                fault_feedback_in := "conveyor_6".fault_feedback_out,
                fault_reset := "reset_button",
                preceeding_sensor := "sensor(4)",
                off_delay := "standard_parameters"."6 meter belt clearance delay",
                system_fault_flag := "system_state".fault_flag,
                "motor+" => "motor+(5)",
                "motor-" => "motor-(5)");
END_REGION

REGION Network 3
   "conveyor_4"(enable_cascade_control := 0,   // "conveyor_control"
                enable_sensor_control := 1,
                enable_on_delay := 0,
                enable_off_delay := 1,
                encoder_A := "encoder_A(4)",
                encoder_B := "encoder_B(4)",
                fault_feedback_in := "conveyor_5".fault_feedback_out,
                fault_reset := "reset_button",
                preceeding_sensor := "sensor(3)",
                off_delay := "standard_parameters"."curved belt clearance delay",
                system_fault_flag := "system_state".fault_flag,
                "motor+" => "motor+(4)",
                "motor-" => "motor-(4)");
END_REGION

REGION Network 4
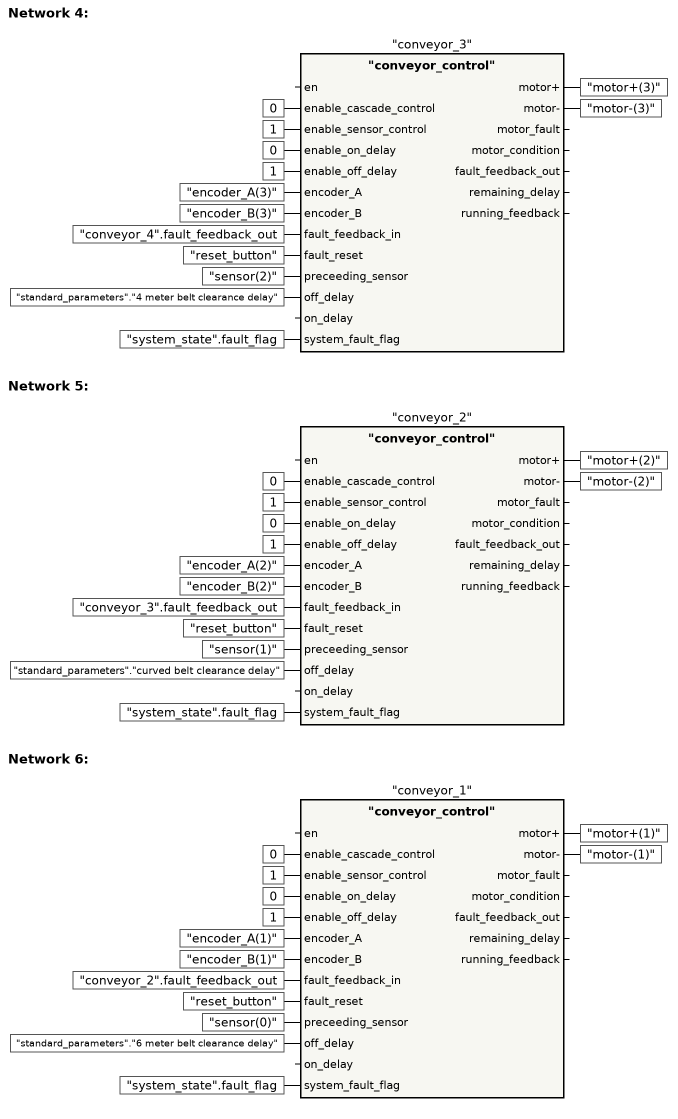
   "conveyor_3"(enable_cascade_control := 0,   // "conveyor_control"
                enable_sensor_control := 1,
                enable_on_delay := 0,
                enable_off_delay := 1,
                encoder_A := "encoder_A(3)",
                encoder_B := "encoder_B(3)",
                fault_feedback_in := "conveyor_4".fault_feedback_out,
                fault_reset := "reset_button",
                preceeding_sensor := "sensor(2)",
                off_delay := "standard_parameters"."4 meter belt clearance delay",
                system_fault_flag := "system_state".fault_flag,
                "motor+" => "motor+(3)",
                "motor-" => "motor-(3)");
END_REGION

REGION Network 5
   "conveyor_2"(enable_cascade_control := 0,   // "conveyor_control"
                enable_sensor_control := 1,
                enable_on_delay := 0,
                enable_off_delay := 1,
                encoder_A := "encoder_A(2)",
                encoder_B := "encoder_B(2)",
                fault_feedback_in := "conveyor_3".fault_feedback_out,
                fault_reset := "reset_button",
                preceeding_sensor := "sensor(1)",
                off_delay := "standard_parameters"."curved belt clearance delay",
                system_fault_flag := "system_state".fault_flag,
                "motor+" => "motor+(2)",
                "motor-" => "motor-(2)");
END_REGION

REGION Network 6
   "conveyor_1"(enable_cascade_control := 0,   // "conveyor_control"
                enable_sensor_control := 1,
                enable_on_delay := 0,
                enable_off_delay := 1,
                encoder_A := "encoder_A(1)",
                encoder_B := "encoder_B(1)",
                fault_feedback_in := "conveyor_2".fault_feedback_out,
                fault_reset := "reset_button",
                preceeding_sensor := "sensor(0)",
                off_delay := "standard_parameters"."6 meter belt clearance delay",
                system_fault_flag := "system_state".fault_flag,
                "motor+" => "motor+(1)",
                "motor-" => "motor-(1)");
END_REGION

REGION Network 7
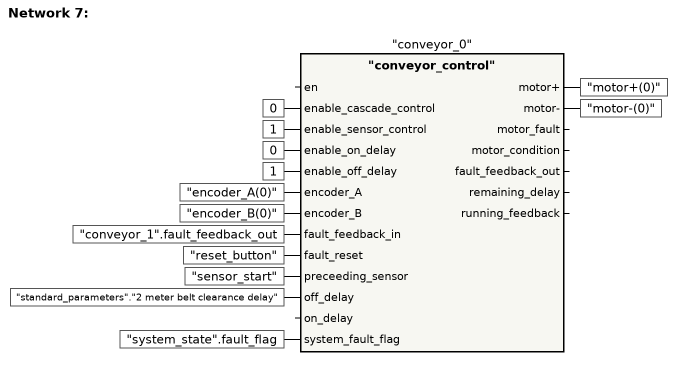
   "conveyor_0"(enable_cascade_control := 0,   // "conveyor_control"
                enable_sensor_control := 1,
                enable_on_delay := 0,
                enable_off_delay := 1,
                encoder_A := "encoder_A(0)",
                encoder_B := "encoder_B(0)",
                fault_feedback_in := "conveyor_1".fault_feedback_out,
                fault_reset := "reset_button",
                preceeding_sensor := "sensor_start",
                off_delay := "standard_parameters"."2 meter belt clearance delay",
                system_fault_flag := "system_state".fault_flag,
                "motor+" => "motor+(0)",
                "motor-" => "motor-(0)");
END_REGION
END_FUNCTION

FUNCTION "MHJ-PLC-Lab-Function-S71500" : Void   // FC9000, SCL
{ S7_Optimized_Access := 'TRUE' }
VERSION : 0.1
   VAR_TEMP
      Value : Byte;
      ForCounter : Int;
   END_VAR
   VAR CONSTANT
      Value_01_DW : DWord := 16#1223_5486;
      Value_02_DW : DWord := 16#A6C9_D1F5;
   END_VAR
BEGIN

   #Value:=PEEK(area := 16#82,
        dbNumber := 0,
        byteOffset := 511);
   #Value := #Value + 1;

   POKE(area := 16#82,
        dbNumber := 0,
        byteOffset := 511,
        value := #Value);

   POKE(area := 16#82,
        dbNumber := 0,
        byteOffset := 1016,
        value := #Value_01_DW);
   POKE(area := 16#82,
        dbNumber := 0,
        byteOffset := 1020,
        value := #Value_02_DW);

   FOR #ForCounter := 0 TO 63 DO
       #Value:=PEEK(area := 16#1,
            dbNumber := 0,
            byteOffset := #ForCounter);
       POKE(area := 16#81,
            dbNumber := 0,
            byteOffset := #ForCounter,
            value := #Value);
   END_FOR;
   #Value := PEEK(area := 16#1,
                  dbNumber := 0,
                  byteOffset := 512);
   POKE(area := 16#82,
        dbNumber := 0,
        byteOffset := 512,
        value := #Value);
END_FUNCTION

ORGANIZATION_BLOCK "Main"   // OB1, FBD, ProgramCycle
TITLE = "Main Program Sweep (Cycle)"
{ S7_Optimized_Access := 'TRUE' }
VERSION : 0.1
   VAR_INPUT
      Initial_Call : Bool;   // Initial call of this OB
      Remanence : Bool;   // =True, if remanent data are available
   END_VAR
BEGIN

REGION Network 1
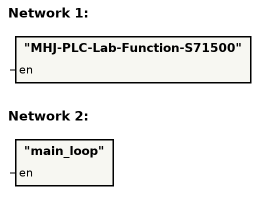
   "MHJ-PLC-Lab-Function-S71500"();
END_REGION

REGION Network 2
   "main_loop"();
END_REGION
END_ORGANIZATION_BLOCK

(* ===== HMI "HMI_RT_2" =====
system functions are stored by id; their names below are inferred from use
connection "HMI_Connection_1": ETHERNET, SMART_S7_1500_OMS

HMI tags "Default tag table"
   "Tag_ScreenNumber" : UInt, internal
   "system state_all conveyors running" : Bool = PLC system_state.all_conveyors_running, 1 s
   "system state_safety delay" : Time = PLC system_state.safety_delay, 1 s

HMI tags "conveyors"
   "conveyor_0" : Int = PLC conveyor_0.motor_condition AT %DB1.DBW0, 100 ms
   "conveyor_1" : Int = PLC conveyor_1.motor_condition, 100 ms
   "conveyor_2" : Int = PLC conveyor_2.motor_condition, 100 ms
   "conveyor_3" : Int = PLC conveyor_3.motor_condition, 100 ms
   "conveyor_4" : Int = PLC conveyor_4.motor_condition, 100 ms
   "conveyor_5" : Int = PLC conveyor_5.motor_condition, 100 ms
   "conveyor_6" : Int = PLC conveyor_6.motor_condition, 100 ms

HMI tags "conveyor time"
   "conveyor_delay_0" : Time = PLC conveyor_0.remaining_delay, 100 ms
   "conveyor_delay_1" : Time = PLC conveyor_1.remaining_delay, 100 ms
   "conveyor_delay_2" : Time = PLC conveyor_2.remaining_delay, 100 ms
   "conveyor_delay_3" : Time = PLC conveyor_3.remaining_delay, 100 ms
   "conveyor_delay_4" : Time = PLC conveyor_4.remaining_delay, 100 ms
   "conveyor_delay_5" : Time = PLC conveyor_5.remaining_delay, 100 ms
   "conveyor_delay_6" : Time = PLC conveyor_6.remaining_delay, 100 ms

HMI tags "system state"
   "system start lamp" : Bool = PLC system_start AT %Q0.3, 100 ms
   "system fault lamp" : Bool = PLC system_fault AT %Q0.4, 100 ms
   "system stop lamp" : Bool = PLC system_stop AT %Q0.5, 100 ms
   "low power mode" : Bool = PLC system_state.low_power_mode, 100 ms
   "safety delay" : Time = PLC system_state.safety_delay, 100 ms

Template "Template_1" 1280x800
   Button "Exit" at 1182,752 size 67x47; TextOff 'Exit'; PictureOff "ExitRuntime_KTP1200_Basic_PN_TR"; PictureOn "ExitRuntime_KTP1200_Basic_PN_TR"
      on Release: StopRuntime(0)
   Button "Template_Button" at 1054,752 size 67x47; TextOff 'Text'
   Button "Template_Button_1" at 926,752 size 67x47; TextOff 'Text'
   Button "Template_Button_2" at 798,752 size 67x47; TextOff 'Text'
   Button "Template_Button_3" at 670,752 size 67x47; TextOff 'Text'
   Button "Template_Button_4" at 542,752 size 67x47; TextOff 'Text'
   Button "Template_Button_5" at 414,752 size 67x47; TextOff 'Text'
   Button "Template_Button_6" at 286,752 size 67x47; TextOff 'Text'
   Button "Alarms" at 158,752 size 67x47; TextOff 'Alarms'; PictureOff "AlarmDisplay_KTP1200_Basic_PN_TR"; PictureOn "AlarmDisplay_KTP1200_Basic_PN_TR"
      on Release: function_ef3f5d25("Alarm window_Unacknowledged", -1)
   Button "Start screen" at 30,752 size 67x47; TextOff 'Start screen'; PictureOff "NavigateHome_KTP1200_Basic_PN_TR"; PictureOn "NavigateHome_KTP1200_Basic_PN_TR"
      on Release: ActivateScreen("Root screen", 0)
   SymbolicIOField "Symbolic_IO_Field_Screen" at 87,9 size 1086x30; TextOff '0'; TextOn '1'; TextList "TextList_ScreenNames"
      ProcessValue <- "Tag_ScreenNumber"
      on Change: ActivateScreenByNumber("Tag_ScreenNumber", 0)
   DateTimeField "HmiScreenItemData" at 1175,24 size 105x24
   DateTimeField "HmiScreenItemData_1" at 1175,0 size 105x24
   GraphicView "Logo" at 0,0 size 85x48; Picture "Logo of HMI_2"

screen "Root screen" 1280x800, template "Template_1"
   on GenerateScreen: SetTag("Tag_ScreenNumber", 1)
   Rectangle "Rectangle_1" at 192,468 size 96x48
      Appearance <- "conveyor_0"
   Rectangle "Rectangle_2" at 289,468 size 288x48
      Appearance <- "conveyor_1"
   Rectangle "Rectangle_3" at 578,468 size 48x48
      Appearance <- "conveyor_2"
   Rectangle "Rectangle_4" at 578,275 size 48x192
      Appearance <- "conveyor_3"
   Rectangle "Rectangle_5" at 192,226 size 96x48
      Appearance <- "conveyor_6"
   Rectangle "Rectangle_6" at 289,226 size 288x48
      Appearance <- "conveyor_5"
   Rectangle "Rectangle_7" at 578,226 size 48x48
      Appearance <- "conveyor_4"
   IOField "I/O field_2" at 193,435 size 96x32; FormatPattern s9999999999
      ProcessValue <- "conveyor_delay_0"
   IOField "I/O field_1" at 384,435 size 96x32; FormatPattern s9999999999
      ProcessValue <- "conveyor_delay_1"
   IOField "I/O field_3" at 626,476 size 96x32; FormatPattern s9999999999
      ProcessValue <- "conveyor_delay_2"
   IOField "I/O field_4" at 626,361 size 96x32; FormatPattern s9999999999
      ProcessValue <- "conveyor_delay_3"
   IOField "I/O field_5" at 626,234 size 96x32; FormatPattern s9999999999
      ProcessValue <- "conveyor_delay_4"
   IOField "I/O field_6" at 384,194 size 96x32; FormatPattern s9999999999
      ProcessValue <- "conveyor_delay_5"
   IOField "I/O field_7" at 192,194 size 96x32; FormatPattern s9999999999
      ProcessValue <- "conveyor_delay_6"
   TextField "Text field_1" at 206,410 size 68x25; Text 'conv_0'
   TextField "Text field_2" at 396,410 size 68x25; Text 'conv_1'
   TextField "Text field_3" at 636,451 size 68x25; Text 'conv_2'
   TextField "Text field_4" at 636,336 size 68x25; Text 'conv_3'
   TextField "Text field_5" at 636,209 size 68x25; Text 'conv_4'
   TextField "Text field_6" at 396,169 size 68x25; Text 'conv_5'
   TextField "Text field_7" at 206,169 size 68x25; Text 'conv_6'
   Rectangle "Rectangle_8" at 193,570 size 96x48
      Appearance <- "system stop lamp"
   Rectangle "Rectangle_9" at 193,620 size 96x48
      Appearance <- "system fault lamp"
   Rectangle "Rectangle_10" at 193,670 size 96x48
      Appearance <- "system start lamp"
   TextField "Text field_8" at 304,680 size 45x25; Text 'start'
   TextField "Text field_9" at 304,632 size 45x25; Text 'fault'
   TextField "Text field_10" at 304,584 size 43x25; Text 'stop'
   Circle "Circle_1" at 513,679 size 48x48
      Appearance <- "low power mode"
   Circle "Circle_2" at 513,620 size 48x48
      Appearance <- "system state_all conveyors running"
   TextField "Text field_11" at 577,574 size 109x25; Text 'safety delay'
   TextField "Text field_12" at 577,632 size 190x25; Text 'all conveyors running'
   TextField "Text field_13" at 577,693 size 148x25; Text 'low power mode'
   IOField "I/O field_8" at 465,570 size 96x32; FormatPattern s9999999999
      ProcessValue <- "safety delay"
      Appearance <- "safety delay"
*)